FUNCTION_BLOCK F_INT_TO_LREAL (* Convert INT to LREAL *)
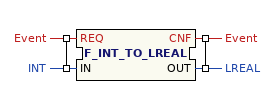
  EVENT_INPUT
    REQ WITH IN; (* Normal Execution Request *)
  END_EVENT
  EVENT_OUTPUT
    CNF WITH OUT; (* Execution Confirmation *)
  END_EVENT
  VAR_INPUT
    IN : INT;
  END_VAR
  VAR_OUTPUT
    OUT : LREAL;
  END_VAR
END_FUNCTION_BLOCK
